# B&R Automation Studio project report1
Automation Studio 4.5.2.102

## Configuration Config1

### Task classes (Cpu.sw)
```
Cyclic#1 (cycle 2000 us, tolerance 0 us):
  ncsdcctrl <- ncsdcctrl.prg
Cyclic#3:
  Program1 <- Program1.prg
Cyclic#4:
  Program2 <- Program2.prg
Cyclic#5:
  Program3 <- Program3.prg
Cyclic#6:
  Program4 <- Program4.prg
DataObjects: Acp10sys
NcDataObjects: acp10etxen <- acp10etxen.dob, gAxis01a <- gAxis01obj.gAxis01a.dob, gAxis01i <- gAxis01obj.gAxis01i.dob, gAxis02a <- gAxis02obj.gAxis02a.dob, gAxis02i <- gAxis02obj.gAxis02i.dob
Binaries: TCData, udbdef, iomap, arconfig, asfw, ashwac, sysconf, User, Role, ashwd, acp10cfg, Acp10map
Libraries: Acp10man, Acp10par, NcGlobal, Acp10sdc, Acp10_MC, brsystem, sys_lib, runtime, AsBrStr, astime, fileio, powerlnk, asieccon
```

### Hardware
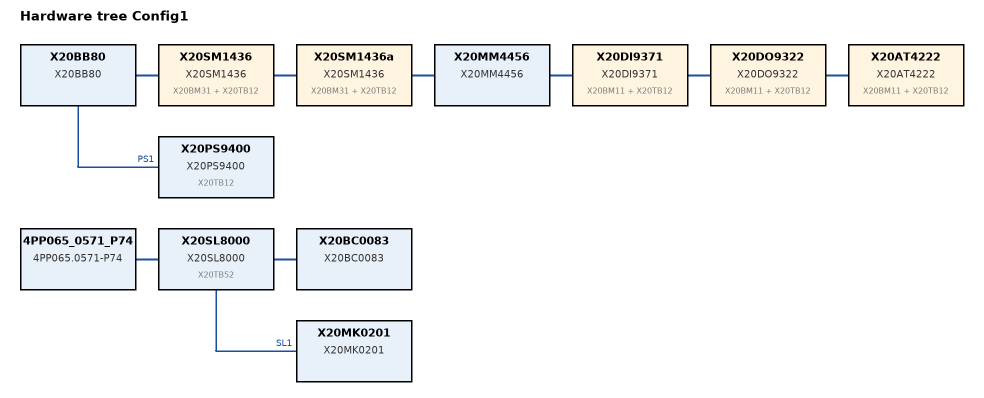
```
4PP065_0571_P74 : 4PP065.0571-P74 v1.1.2.0
  Connector IF5:
    ActivateDevice = 1
    Mode = Manual
    InternetAddress = 10.0.1.10
    SubnetMask = 255.255.255.0
  ConfigurationID = labBR
  TimerDeviceType = EPLX2X
  TimerDevice = 4PP065_0571_P74.IF4
  TaskClassIdleTime = 2000
  Cyclic1Duration = 2000
  Cyclic1Tolerance = 0
  Cyclic1Output = 1
X20AT4222 : X20AT4222 v1.2.3.0  [SS1 -> X20TB12e.SS; SL -> X20BM11b.SL1]
X20BB80 : X20BB80 v1.0.2.0
X20BC0083 : X20BC0083 v2.9.0.0  [PLK1 -> X20SL8000.PLK2 [Cable Type=PowerlinkCable, Length=10, Version=1.0.0.2]; SL -> X20BB80.SL1]
X20BM11 : X20BM11 v1.0.0.1  [X2X1 -> X20MM4456.X2X2]
X20BM11a : X20BM11 v1.0.0.1  [X2X1 -> X20BM11.X2X2]
X20BM11b : X20BM11 v1.0.0.1  [X2X1 -> X20BM11a.X2X2]
X20BM31 : X20BM31 v1.0.0.1  [X2X1 -> X20BB80.IF1]
X20BM31a : X20BM31 v1.0.0.1  [X2X1 -> X20BM31.X2X2]
X20DI9371 : X20DI9371 v1.0.2.0  [SS1 -> X20TB12c.SS; SL -> X20BM11.SL1]
X20DO9322 : X20DO9322 v1.0.3.0  [SS1 -> X20TB12d.SS; SL -> X20BM11a.SL1]
X20MK0201 : X20MK0201 v1.0.0.0  [SL -> X20SL8000.SL1]
X20MM4456 : X20MM4456 v1.4.0.0  [X2X1 -> X20BM31a.X2X2]
X20PS9400 : X20PS9400 v1.0.2.4  [SS1 -> X20TB12.SS; PS -> X20BB80.PS1]
X20SL8000 : X20SL8000 v1.6.5.1  [PLK1 -> 4PP065_0571_P74.IF4 [Cable Type=PowerlinkCable, Length=10, Version=1.0.0.2]; PLK2 -> X20BC0083.PLK1 [Cable Type=PowerlinkCable, Length=10, Version=1.0.0.2]; SS1 -> X20TB52.SS]
  SafeProject = SafeLOGIC-1
X20SM1436 : X20SM1436 v1.4.2.1  [SS1 -> X20TB12a.SS; SL -> X20BM31.SL1]
X20SM1436a : X20SM1436 v1.4.2.1  [SS1 -> X20TB12b.SS; SL -> X20BM31a.SL1]
X20TB12 : X20TB12 v1.0.0.0
X20TB12a : X20TB12 v1.0.0.0
X20TB12b : X20TB12 v1.0.0.0
X20TB12c : X20TB12 v1.0.0.0
X20TB12d : X20TB12 v1.0.0.0
X20TB12e : X20TB12 v1.0.0.0
X20TB52 : X20TB52 v1.0.0.1
```

### IoMap.iom - 4PP065_0571_P74/IoMap.iom
```iecst
VAR_CONFIG
	Cyclic#1.gAxis01_DrvIf.iLifeCnt AT %IB."X20SM1436".LifeCnt;
	Cyclic#1.gAxis01_DrvIf.iDrvOK AT %IX."X20SM1436".DrvOk01;
	Cyclic#1.gAxis01_DrvIf.oBoostCurrent AT %QX."X20SM1436".BoostCurrent01;
	Cyclic#1.gAxis01_DrvIf.oStandStillCurrent AT %QX."X20SM1436".StandstillCurrent01;
	Cyclic#1.gAxis01_DrvIf.oSetTime AT %QW."X20SM1436".SetTime01;
	Cyclic#1.gAxis01_MotorStep0 AT %QW."X20SM1436".Motor1Step0;
	Cyclic#1.gAxis01_DiDoIf.iLifeCntDriveEnable AT %IB."X20SM1436".LifeCnt;
	Cyclic#1.gAxis01_DiDoIf.iLifeCntDriveReady AT %IB."X20SM1436".LifeCnt;
	Cyclic#1.gAxis01_DiDoIf.iDriveReady AT %IX."X20SM1436".DrvOk01;
	Cyclic#1.gAxis01_DiDoIf.oDriveEnable AT %QX."X20SM1436".DriveEnable01;
	Cyclic#1.gAxis01_EncIf1.iLifeCnt AT %IB."X20SM1436".LifeCnt;
	Cyclic#1.gAxis01_EncIf1.iEncOK AT %IX."X20SM1436".EncOk01;
	Cyclic#1.gAxis01_EncIf1.iActPos AT %IW."X20SM1436".ActPos01;
	Cyclic#1.gAxis01_EncIf1.iRefPulsePos AT %IW."X20SM1436".RefPulsePos01;
	Cyclic#1.gAxis01_EncIf1.iRefPulseCnt AT %IB."X20SM1436".RefPulseCnt01;
	Cyclic#1.gAxis01_EncIf1.iActTime AT %IW."X20SM1436".ActTime01;
	Cyclic#1.gAxis02_DrvIf.iLifeCnt AT %IB."X20SM1436a".LifeCnt;
	Cyclic#1.gAxis02_DrvIf.iDrvOK AT %IX."X20SM1436a".DrvOk01;
	Cyclic#1.gAxis02_DrvIf.oBoostCurrent AT %QX."X20SM1436a".BoostCurrent01;
	Cyclic#1.gAxis02_DrvIf.oStandStillCurrent AT %QX."X20SM1436a".StandstillCurrent01;
	Cyclic#1.gAxis02_DrvIf.oSetTime AT %QW."X20SM1436a".SetTime01;
	Cyclic#1.gAxis02_MotorStep0 AT %QW."X20SM1436a".Motor1Step0;
	Cyclic#1.gAxis02_DiDoIf.iLifeCntDriveEnable AT %IB."X20SM1436a".LifeCnt;
	Cyclic#1.gAxis02_DiDoIf.iLifeCntDriveReady AT %IB."X20SM1436a".LifeCnt;
	Cyclic#1.gAxis02_DiDoIf.iDriveReady AT %IX."X20SM1436a".DrvOk01;
	Cyclic#1.gAxis02_DiDoIf.oDriveEnable AT %QX."X20SM1436a".DriveEnable01;
	Cyclic#1.gAxis02_EncIf1.iLifeCnt AT %IB."X20SM1436a".LifeCnt;
	Cyclic#1.gAxis02_EncIf1.iEncOK AT %IX."X20SM1436a".EncOk01;
	Cyclic#1.gAxis02_EncIf1.iActPos AT %IW."X20SM1436a".ActPos01;
	Cyclic#1.gAxis02_EncIf1.iRefPulsePos AT %IW."X20SM1436a".RefPulsePos01;
	Cyclic#1.gAxis02_EncIf1.iRefPulseCnt AT %IB."X20SM1436a".RefPulseCnt01;
	Cyclic#1.gAxis02_EncIf1.iActTime AT %IW."X20SM1436a".ActTime01;
	::led1 AT %QX."X20DO9322".DigitalOutput02;
	::led2 AT %QX."X20DO9322".DigitalOutput03;
	::led3 AT %QX."X20DO9322".DigitalOutput04;
	::led4 AT %QX."X20DO9322".DigitalOutput05;
END_VAR
```

### Acp10map.ncm - 4PP065_0571_P74/Motion/Acp10map.ncm
```
NcMapping (NcSwId=Acp10)
  NcObject gAxis01 (ModuleId=X20SM1436, ModuleAddress=SDC_IF1.ST1, Type=ncAXIS, Channel=1, AcoposSimulation=Off, InitParameter=gAxis01i, AcoposParameter=gAxis01a, Disabled=FALSE, ModuleDisabled=FALSE)
  NcObject gAxis02 (ModuleId=X20SM1436a, ModuleAddress=SDC_IF1.ST2, Type=ncAXIS, Channel=1, AcoposSimulation=Off, InitParameter=gAxis02i, AcoposParameter=gAxis02a, Disabled=FALSE, ModuleDisabled=FALSE)
```

## Logical view

### Global.var - Global variables
```iecst
VAR
	gAxis01 : ACP10AXIS_typ;
	gAxis01_HW : SdcHwCfg_typ := (0);
	gAxis01_DrvIf : SdcDrvIf16_typ := (0);
	gAxis01_EncIf1 : SdcEncIf16_typ := (0);
	gAxis01_DiDoIf : SdcDiDoIf_typ := (0);
	gAxis01_MotorStep0 : INT := (0);
	gAxis02 : ACP10AXIS_typ;
	gAxis02_HW : SdcHwCfg_typ := (0);
	gAxis02_DrvIf : SdcDrvIf16_typ := (0);
	gAxis02_EncIf1 : SdcEncIf16_typ := (0);
	gAxis02_DiDoIf : SdcDiDoIf_typ := (0);
	gAxis02_MotorStep0 : INT := (0);
	led1 : {REDUND_UNREPLICABLE} BOOL;
	led2 : {REDUND_UNREPLICABLE} BOOL;
	led3 : {REDUND_UNREPLICABLE} BOOL;
	led4 : {REDUND_UNREPLICABLE} BOOL;
END_VAR
```

### Program Logical/ncsdcctrl (IEC)

#### ncsdcctrlCyclic.st
```iecst
PROGRAM _CYCLIC

(* ### BEGIN gAxis01 ### *)

(* life counter emulation of digital inputs *)
      gAxis01_DiDoIf.iLifeCntReference := gAxis01_DiDoIf.iLifeCntReference + 1;
      gAxis01_DiDoIf.iLifeCntNegHwEnd  := gAxis01_DiDoIf.iLifeCntNegHwEnd  + 1;
      gAxis01_DiDoIf.iLifeCntPosHwEnd  := gAxis01_DiDoIf.iLifeCntPosHwEnd  + 1;

(* default function model of ACOPOSmicro: convert absolute steps to delta steps - overflow save delta calculation *)
      gAxis01_MotorStep0 := gAxis01_DrvIf.oSetPos - gAxis01_oSetPosOld;
      gAxis01_oSetPosOld := gAxis01_DrvIf.oSetPos;

(* ### END gAxis01 ### *)

(* ### BEGIN gAxis02 ### *)

(* life counter emulation of digital inputs *)
      gAxis02_DiDoIf.iLifeCntReference := gAxis02_DiDoIf.iLifeCntReference + 1;
      gAxis02_DiDoIf.iLifeCntNegHwEnd  := gAxis02_DiDoIf.iLifeCntNegHwEnd  + 1;
      gAxis02_DiDoIf.iLifeCntPosHwEnd  := gAxis02_DiDoIf.iLifeCntPosHwEnd  + 1;

(* default function model of ACOPOSmicro: convert absolute steps to delta steps - overflow save delta calculation *)
      gAxis02_MotorStep0 := gAxis02_DrvIf.oSetPos - gAxis02_oSetPosOld;
      gAxis02_oSetPosOld := gAxis02_DrvIf.oSetPos;

(* ### END gAxis02 ### *)

END_PROGRAM
```

#### ncsdcctrlInit.st
```iecst
PROGRAM _INIT

(* ### BEGIN gAxis01 ### *)

(* initialize general interfaces *)
      gAxis01.size := gAxis01.size;
      gAxis01_HW.DrvIf_Typ := ncSDC_DRVSM16;
      brsstrcpy( ADR(gAxis01_HW.DrvIf_Name[0]), ADR('gAxis01_DrvIf') );
      gAxis01_HW.DiDoIf_Typ := ncSDC_DIDO;
      brsstrcpy( ADR(gAxis01_HW.DiDoIf_Name[0]), ADR('gAxis01_DiDoIf') );
      gAxis01_HW.EncIf1_Typ := ncSDC_ENC16;
      brsstrcpy( ADR(gAxis01_HW.EncIf1_Name[0]), ADR('gAxis01_EncIf1') );
      gAxis01_EncIf1.iLifeCnt := gAxis01_EncIf1.iLifeCnt;

(* initialize old-value for delta step calculation *)
      gAxis01_oSetPosOld := gAxis01_DrvIf.oSetPos;

(* ### END gAxis01 ### *)

(* ### BEGIN gAxis02 ### *)

(* initialize general interfaces *)
      gAxis02.size := gAxis02.size;
      gAxis02_HW.DrvIf_Typ := ncSDC_DRVSM16;
      brsstrcpy( ADR(gAxis02_HW.DrvIf_Name[0]), ADR('gAxis02_DrvIf') );
      gAxis02_HW.DiDoIf_Typ := ncSDC_DIDO;
      brsstrcpy( ADR(gAxis02_HW.DiDoIf_Name[0]), ADR('gAxis02_DiDoIf') );
      gAxis02_HW.EncIf1_Typ := ncSDC_ENC16;
      brsstrcpy( ADR(gAxis02_HW.EncIf1_Name[0]), ADR('gAxis02_EncIf1') );
      gAxis02_EncIf1.iLifeCnt := gAxis02_EncIf1.iLifeCnt;

(* initialize old-value for delta step calculation *)
      gAxis02_oSetPosOld := gAxis02_DrvIf.oSetPos;

(* ### END gAxis02 ### *)

END_PROGRAM
```

### Program Logical/Program1 (ANSIC)

#### Variables.var
```iecst
VAR
	i : {REDUND_UNREPLICABLE} INT;
END_VAR
```

#### Main.c
```c
#include <bur/plctypes.h>

#ifdef _DEFAULT_INCLUDES
	#include <AsDefault.h>
#endif

void _INIT ProgramInit(void)
{
	led1 = 0;
	/*led2 = 0;
	led3 = 0;
	led4 = 0;
	i = 0;*/
}

void _CYCLIC ProgramCyclic(void)
{
	led1 = !led1;
	/*if(i%8==0){
		led1 = !led1;
	}
	if(i%8 == 2){
		led2 = !led2;
	}
	if(i%8 == 4){
		led3 = !led3;
	}
	if(i%8 == 6){
		led4 = !led4;
	}
	i++;*/
}

void _EXIT ProgramExit(void)
{

}
```

### Program Logical/Program2 (ANSIC)

#### Main.c
```c
#include <bur/plctypes.h>

#ifdef _DEFAULT_INCLUDES
	#include <AsDefault.h>
#endif

void _INIT ProgramInit(void)
{
	led2 = 0;
}

void _CYCLIC ProgramCyclic(void)
{
	led2 = !led2;
}

void _EXIT ProgramExit(void)
{

}
```

### Program Logical/Program3 (ANSIC)

#### Main.c
```c
#include <bur/plctypes.h>

#ifdef _DEFAULT_INCLUDES
	#include <AsDefault.h>
#endif

void _INIT ProgramInit(void)
{
	led3 = 0;
}

void _CYCLIC ProgramCyclic(void)
{
	led3 = !led3;
}

void _EXIT ProgramExit(void)
{

}
```

### Program Logical/Program4 (ANSIC)

#### Main.c
```c
#include <bur/plctypes.h>

#ifdef _DEFAULT_INCLUDES
	#include <AsDefault.h>
#endif

void _INIT ProgramInit(void)
{
	led4 = 0;
}

void _CYCLIC ProgramCyclic(void)
{
	led4 = !led4;
}

void _EXIT ProgramExit(void)
{

}
```

Listed in the project but not available here: Logical/Global.typ, Logical/Libraries, Logical/acp10etxen, Logical/gAxis01obj, Logical/gAxis02obj
